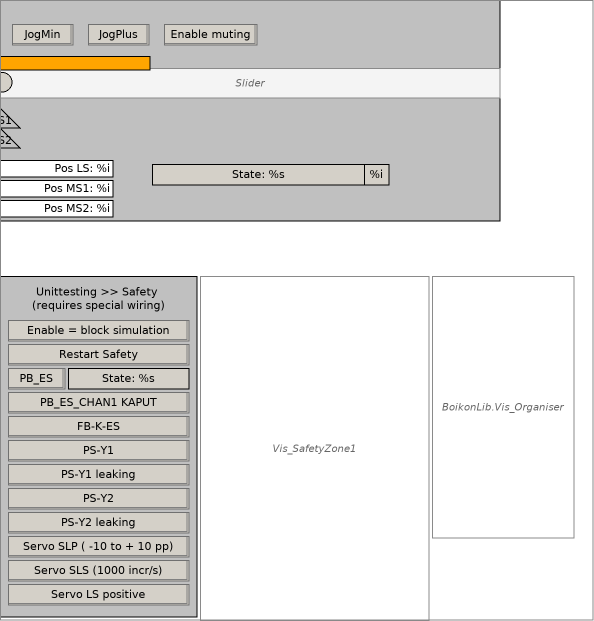
VISUALIZATION Vis_Test  // 594x621
    Rectangle (0,0 500x221)
    Slider (0,68 500x30), variable: UnitTesting.Sft_LS_PosBox, scale 0..485
    Rectangle (0,56 150x14)
        p3560616238: UnitTesting.Sft_LS_PosBox + 0
    Polyline (-20,128) (0,108) (20,128) (-20,128), "MS1", colour toggle: UnitTesting.Qsf_LS_Muting1
        p3560616238: UnitTesting.Sft_LS_PosMS1 + 0
    Polyline (-20,148) (0,128) (20,148) (-20,148), "MS2", colour toggle: UnitTesting.Qsf_LS_Muting2
        p3560616238: UnitTesting.Sft_LS_PosMS2 + 0
    Line (0,20) (0,152), colour toggle: UnitTesting.Qsf_LS_OSSD
        p3560616238: UnitTesting.Sft_LS_PosLS
    Rectangle (0,160 113x17), "Pos LS: %i", text variable: UnitTesting.Sft_LS_PosLS
        OnMouseClick: write the text variable via Edit
    Rectangle (0,180 113x17), "Pos MS1: %i", text variable: UnitTesting.Sft_LS_PosMS1
        OnMouseClick: write the text variable via Edit
    Rectangle (0,200 113x17), "Pos MS2: %i", text variable: UnitTesting.Sft_LS_PosMS2
        OnMouseClick: write the text variable via Edit
    Frame (200,276 229x345)
        shows Vis_SafetyZone1(I_Title := 'SafetyZone 1', IO_SafetyLogic := MAIN.General.SafetyController)
    Button (12,24 61x21), "JogMin"
        tap UnitTesting.Sft_LS_JogBoxMin
    Button (88,24 61x21), "JogPlus"
        tap UnitTesting.Sft_LS_JogBoxPlus
    Rectangle (0,276 197x341)
    Button (8,416 181x21), "FB-K-ES", pressed state: UnitTesting.Sft_FB_K_ES_OK
        toggle UnitTesting.Sft_FB_K_ES_OK
    Button (8,440 181x21), "PS-Y1", pressed state: UnitTesting.Sft_Y_FB1
        toggle UnitTesting.Sft_Y_FB1
    Button (8,488 181x21), "PS-Y2", pressed state: UnitTesting.Sft_Y_FB2
        toggle UnitTesting.Sft_Y_FB2
    Button (8,368 57x21), "PB_ES", pressed state: UnitTesting.Sft_PB_ES
        toggle UnitTesting.Sft_PB_ES
    Button (8,320 181x21), "Enable = block simulation", pressed state: UnitTesting.Sft_EnableSafetyTest
        toggle UnitTesting.Sft_EnableSafetyTest
    Button (8,464 181x21), "PS-Y1 leaking", pressed state: UnitTesting.Sft_Y1_Leaking
        toggle UnitTesting.Sft_Y1_Leaking
    Button (8,512 181x21), "PS-Y2 leaking", pressed state: UnitTesting.Sft_Y2_Leaking
        toggle UnitTesting.Sft_Y2_Leaking
    Rectangle (0,276 197x45), "Unittesting >> Safety (requires special wiring)"
    Button (8,536 181x21), "Servo SLP ( -10 to + 10 pp)", pressed state: UnitTesting.Qsf_K_EnableSafePosition
        toggle UnitTesting.Qsf_K_EnableSafePosition
    Button (8,560 181x21), "Servo SLS (1000 incr/s)", pressed state: UnitTesting.Qsf_K_EnableSafeSpeed
        toggle UnitTesting.Qsf_K_EnableSafeSpeed
    Button (8,584 181x21), "Servo LS positive", pressed state: UnitTesting.LS_Positive.I_K_State
        toggle UnitTesting.LS_Positive.I_K_State
    Button (8,344 181x21), "Restart Safety"
        tap UnitTesting.Sft_PB_IllegalRestart
    Button (164,24 93x21), "Enable muting"
        toggle MAIN.General.SafetyController.I_K_EnableLsRejectMuting
    Rectangle (152,164 213x21), "State: %s", text variable: MAIN.General.SafetyController.LS_Entry1._HM_State
    Rectangle (364,164 25x21), "%i", text variable: MAIN.General.SafetyController.LS_Entry1._HM_State
    Ellipse (-8,72 20x20), colour toggle: MAIN.General.SafetyController.LS_Entry1.HMI.STS.StateMuted
        p3560616238: UnitTesting.Sft_LS_PosLS
    Rectangle (68,368 121x21), "State: %s", text variable: MAIN.General.SafetyController.PB_ES_MainCabinet._HM_State
    Button (8,392 181x21), "PB_ES_CHAN1 KAPUT"
        toggle UnitTesting.Sft_PB_ES_Chan1Broken
    Frame (432,276 142x262)
        shows BoikonLib.Vis_Organiser(I_UnitName := 'Organiser'', IO_cntrl_Organiser := MAIN.Organiser)
END_VISUALIZATION

(* stored: Version 1.1.0.1
   Visu Vis_Test: Id {2b9ff988-6909-4a59-be43-59f20b9fe604} *)
